PROGRAM B_2_2_PRG_Fault_Station_2
VAR_INPUT
	
	i										: INT;
	
END_VAR

VAR_IN_OUT
	aAlarms  								: ARRAY[0..3] OF ST_Events;
END_VAR

a_ACT_FaultTrig();

(************************************** Faults reset **********************************************)
IF   stButtonsLamps.bResetButtonFallingEdge THEN 
	FOR i := 0 TO 127 DO
		GVL_MASTER.stAlarms[2].aEventFlags[i] := FALSE;
	END_FOR
END_IF
//===============================================================
//Initialize event texts on first scan
IF NOT GVL_MASTER.stAlarms[2].bEventTextsSet THEN
	b_MET_SetEventTexts();
	GVL_MASTER.stAlarms[2].bEventTextsSet := TRUE;
END_IF


(***************************************************************************************************)
//Immediate fault
GVL_MASTER.stAlarms[2].bImmediateFault := FALSE;
FOR i := 0 TO 32DO
	GVL_MASTER.stAlarms[2].bImmediateFault := GVL_MASTER.stAlarms[2].bImmediateFault OR GVL_MASTER.stAlarms[2].aEventFlags[i];
END_FOR

//Cycle stop fault
GVL_MASTER.stAlarms[2].bCycleStopFault := FALSE;
FOR i := 33 TO 79 DO
	GVL_MASTER.stAlarms[2].bCycleStopFault := GVL_MASTER.stAlarms[2].bCycleStopFault OR GVL_MASTER.stAlarms[2].aEventFlags[i];
END_FOR

//Cycle stop REQUEST
GVL_MASTER.stAlarms[2].bCycleStopRequest := FALSE;
FOR i := 80 TO 99 DO
	GVL_MASTER.stAlarms[2].bCycleStopRequest := GVL_MASTER.stAlarms[2].bCycleStopRequest OR GVL_MASTER.stAlarms[2].aEventFlags[i];
END_FOR

ACTION a_ACT_FaultTrig:

/////////////////////////////////////////////////////////////////////////////////////Immediate Faults 0-32////////////////////////////////////////////////////////////////////////////////////

//Immediate Fault
GVL_MASTER.stAlarms[2].aEventTimers[0]
(IN := ,PT:= T#500MS );
IF GVL_MASTER.stAlarms[2].aEventTimers[0].Q  THEN 
	GVL_MASTER.stAlarms[2].aEventFlags[0] := TRUE;
END_IF

/////////////////////////////////////////////////////////////////////////////////////Cycle stop faults 33-79////////////////////////////////////////////////////////////////////////////////////

////Cycle stop fault
GVL_MASTER.stAlarms[2].aEventTimers[33]
(IN := ,PT:= T#500MS );
IF GVL_MASTER.stAlarms[2].aEventTimers[33].Q THEN 
	GVL_MASTER.stAlarms[2].aEventFlags[33] := TRUE;
END_IF

/////////////////////////////////////////////////////////////////////////////////////Cycle stop Requests 80-99////////////////////////////////////////////////////////////////////////////////////

////Cycle stop Request
GVL_MASTER.stAlarms[2].aEventTimers[80]
(IN := ,PT:= T#500MS );
IF GVL_MASTER.stAlarms[2].aEventTimers[80].Q THEN 
	GVL_MASTER.stAlarms[2].aEventFlags[80] := TRUE;
END_IF
END_ACTION

METHOD b_MET_SetEventTexts : BOOL
VAR_INPUT
END_VAR
/////////////////////////////////////////////////////////////////////////////////////Immediate Faults 0-32////////////////////////////////////////////////////////////////////////////////////

GVL_MASTER.stAlarms[2].aEventTexts[0] := 'Station 2 - Immediate Fault';
GVL_MASTER.stAlarms[2].aEventTexts[1] := '';
GVL_MASTER.stAlarms[2].aEventTexts[2] := '';
GVL_MASTER.stAlarms[2].aEventTexts[4] := '';
GVL_MASTER.stAlarms[2].aEventTexts[5] := '';
GVL_MASTER.stAlarms[2].aEventTexts[6] := '';
GVL_MASTER.stAlarms[2].aEventTexts[7] := '';
GVL_MASTER.stAlarms[2].aEventTexts[8] := '';
GVL_MASTER.stAlarms[2].aEventTexts[9] := '';
GVL_MASTER.stAlarms[2].aEventTexts[10] := ''; 
GVL_MASTER.stAlarms[2].aEventTexts[11] := ''; 
GVL_MASTER.stAlarms[2].aEventTexts[12] := '';
GVL_MASTER.stAlarms[2].aEventTexts[13] := '';
GVL_MASTER.stAlarms[2].aEventTexts[14] := '';
GVL_MASTER.stAlarms[2].aEventTexts[15] := '';
GVL_MASTER.stAlarms[2].aEventTexts[16] := '';
GVL_MASTER.stAlarms[2].aEventTexts[17] := '';
GVL_MASTER.stAlarms[2].aEventTexts[18] := '';
GVL_MASTER.stAlarms[2].aEventTexts[19] := '';
GVL_MASTER.stAlarms[2].aEventTexts[20] := '';
GVL_MASTER.stAlarms[2].aEventTexts[21] := '';
GVL_MASTER.stAlarms[2].aEventTexts[22] := '';
GVL_MASTER.stAlarms[2].aEventTexts[23] := '';
GVL_MASTER.stAlarms[2].aEventTexts[24] := '';
GVL_MASTER.stAlarms[2].aEventTexts[25] := '';
GVL_MASTER.stAlarms[2].aEventTexts[26] := '';
GVL_MASTER.stAlarms[2].aEventTexts[27] := '';
GVL_MASTER.stAlarms[2].aEventTexts[28] := '';
GVL_MASTER.stAlarms[2].aEventTexts[29] := '';
GVL_MASTER.stAlarms[2].aEventTexts[30] := '';
GVL_MASTER.stAlarms[2].aEventTexts[31] := '';
GVL_MASTER.stAlarms[2].aEventTexts[32] := '';

/////////////////////////////////////////////////////////////////////////////////////Cycle stop faults 33-79////////////////////////////////////////////////////////////////////////////////////

GVL_MASTER.stAlarms[2].aEventTexts[33] := 'Cycle stop fault';
GVL_MASTER.stAlarms[2].aEventTexts[34] := '';
GVL_MASTER.stAlarms[2].aEventTexts[35] := '';
GVL_MASTER.stAlarms[2].aEventTexts[36] := '';
GVL_MASTER.stAlarms[2].aEventTexts[37] := '';
GVL_MASTER.stAlarms[2].aEventTexts[38] := '';
GVL_MASTER.stAlarms[2].aEventTexts[39] := '';
GVL_MASTER.stAlarms[2].aEventTexts[40] := '';
GVL_MASTER.stAlarms[2].aEventTexts[41] := '';
GVL_MASTER.stAlarms[2].aEventTexts[42] := '';
GVL_MASTER.stAlarms[2].aEventTexts[43] := '';
GVL_MASTER.stAlarms[2].aEventTexts[44] := '';
GVL_MASTER.stAlarms[2].aEventTexts[45] := '';
GVL_MASTER.stAlarms[2].aEventTexts[46] := '';
GVL_MASTER.stAlarms[2].aEventTexts[47] := '';
GVL_MASTER.stAlarms[2].aEventTexts[48] := '';
GVL_MASTER.stAlarms[2].aEventTexts[49] := '';
GVL_MASTER.stAlarms[2].aEventTexts[50] := '';
GVL_MASTER.stAlarms[2].aEventTexts[51] := '';
GVL_MASTER.stAlarms[2].aEventTexts[52] := '';
GVL_MASTER.stAlarms[2].aEventTexts[53] := '';
GVL_MASTER.stAlarms[2].aEventTexts[54] := '';
GVL_MASTER.stAlarms[2].aEventTexts[55] := '';
GVL_MASTER.stAlarms[2].aEventTexts[56] := '';
GVL_MASTER.stAlarms[2].aEventTexts[57] := '';
GVL_MASTER.stAlarms[2].aEventTexts[58] := '';
GVL_MASTER.stAlarms[2].aEventTexts[59] := '';
GVL_MASTER.stAlarms[2].aEventTexts[60] := '';
GVL_MASTER.stAlarms[2].aEventTexts[61] := '';
GVL_MASTER.stAlarms[2].aEventTexts[62] := '';
GVL_MASTER.stAlarms[2].aEventTexts[63] := '';
GVL_MASTER.stAlarms[2].aEventTexts[64] := '';
GVL_MASTER.stAlarms[2].aEventTexts[65] := '';
GVL_MASTER.stAlarms[2].aEventTexts[66] := '';
GVL_MASTER.stAlarms[2].aEventTexts[67] := '';
GVL_MASTER.stAlarms[2].aEventTexts[68] := '';
GVL_MASTER.stAlarms[2].aEventTexts[69] := '';
GVL_MASTER.stAlarms[2].aEventTexts[70] := '';
GVL_MASTER.stAlarms[2].aEventTexts[71] := '';
GVL_MASTER.stAlarms[2].aEventTexts[73] := '';
GVL_MASTER.stAlarms[2].aEventTexts[74] := '';
GVL_MASTER.stAlarms[2].aEventTexts[75] := '';
GVL_MASTER.stAlarms[2].aEventTexts[76] := '';
GVL_MASTER.stAlarms[2].aEventTexts[77] := '';
GVL_MASTER.stAlarms[2].aEventTexts[78] := '';
GVL_MASTER.stAlarms[2].aEventTexts[79] := '';

/////////////////////////////////////////////////////////////////////////////////////Cycle stop Requests 80-99////////////////////////////////////////////////////////////////////////////////////


GVL_MASTER.stAlarms[2].aEventTexts[80] := 'Cycle stop Request';
GVL_MASTER.stAlarms[2].aEventTexts[81] := '';
GVL_MASTER.stAlarms[2].aEventTexts[82] := '';
GVL_MASTER.stAlarms[2].aEventTexts[83] := '';
GVL_MASTER.stAlarms[2].aEventTexts[84] := '';
GVL_MASTER.stAlarms[2].aEventTexts[85] := '';
GVL_MASTER.stAlarms[2].aEventTexts[86] := '';
GVL_MASTER.stAlarms[2].aEventTexts[87] := ''; 
GVL_MASTER.stAlarms[2].aEventTexts[88] := '';
GVL_MASTER.stAlarms[2].aEventTexts[89] := '';
GVL_MASTER.stAlarms[2].aEventTexts[90] := '';
GVL_MASTER.stAlarms[2].aEventTexts[91] := '';
GVL_MASTER.stAlarms[2].aEventTexts[92] := '';
GVL_MASTER.stAlarms[2].aEventTexts[93] := '';
GVL_MASTER.stAlarms[2].aEventTexts[94] := '';
GVL_MASTER.stAlarms[2].aEventTexts[95] := '';
GVL_MASTER.stAlarms[2].aEventTexts[96] := '';
GVL_MASTER.stAlarms[2].aEventTexts[97] := '';
GVL_MASTER.stAlarms[2].aEventTexts[98] := '';
GVL_MASTER.stAlarms[2].aEventTexts[99] := '';
END_METHOD

END_PROGRAM

(* stored: Version 1.1.0.1, ProductVersion 3.1.4024.13
   POU B_2_2_PRG_Fault_Station_2: Id {a33a6e60-b086-4a07-8116-db1a5f3fb58c}, SpecialFunc None
   Action a_ACT_FaultTrig: Id {df2c7efb-00a9-46e6-b488-a0031ee3b2f4}
   Method b_MET_SetEventTexts: Id {9c3d2989-b33a-4165-8063-77f9f38f13b9} *)
